(* PLC project SafeLOGIC, BrAutomation SafeDESIGNER  5.24.1.0 *)
(* stored: companyURL http://www.br-automation.com, creationDateTime Tue Nov 25 17:14:16 2025 *)

PROGRAM PARA_INT

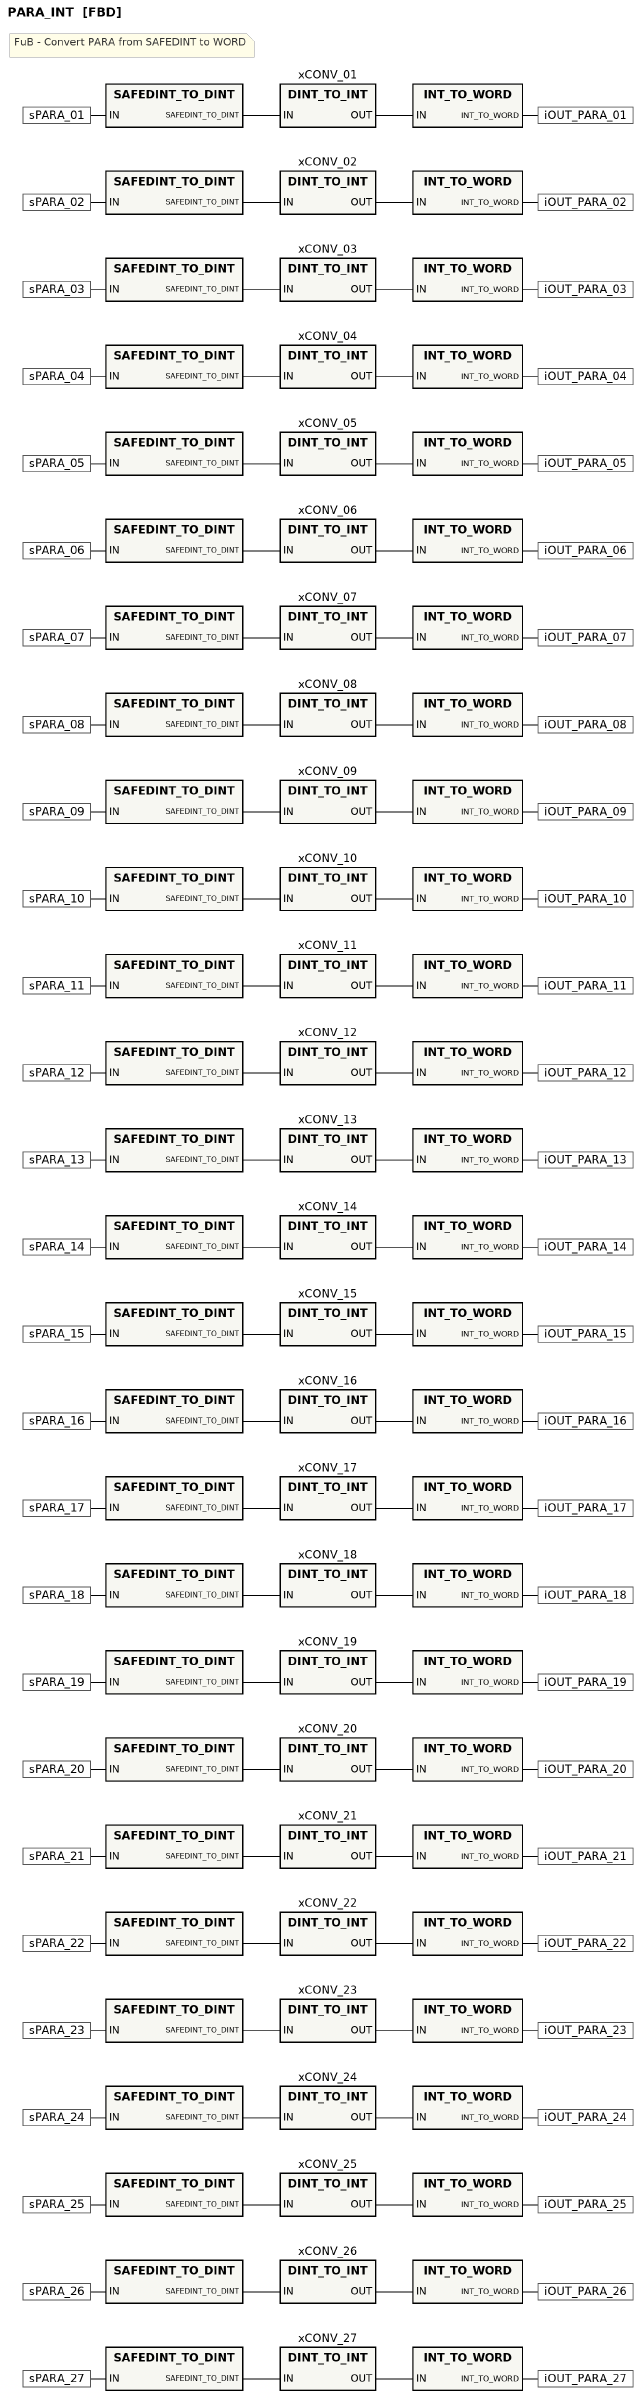
(* FBD diagram, written out as Structured Text *)
(* FuB - Convert PARA from SAFEDINT to WORD *)
xCONV_01(IN := SAFEDINT_TO_DINT(sPARA_01));
iOUT_PARA_01 := INT_TO_WORD(xCONV_01.OUT);
xCONV_02(IN := SAFEDINT_TO_DINT(sPARA_02));
iOUT_PARA_02 := INT_TO_WORD(xCONV_02.OUT);
xCONV_03(IN := SAFEDINT_TO_DINT(sPARA_03));
iOUT_PARA_03 := INT_TO_WORD(xCONV_03.OUT);
xCONV_04(IN := SAFEDINT_TO_DINT(sPARA_04));
iOUT_PARA_04 := INT_TO_WORD(xCONV_04.OUT);
xCONV_05(IN := SAFEDINT_TO_DINT(sPARA_05));
iOUT_PARA_05 := INT_TO_WORD(xCONV_05.OUT);
xCONV_06(IN := SAFEDINT_TO_DINT(sPARA_06));
iOUT_PARA_06 := INT_TO_WORD(xCONV_06.OUT);
xCONV_07(IN := SAFEDINT_TO_DINT(sPARA_07));
iOUT_PARA_07 := INT_TO_WORD(xCONV_07.OUT);
xCONV_08(IN := SAFEDINT_TO_DINT(sPARA_08));
iOUT_PARA_08 := INT_TO_WORD(xCONV_08.OUT);
xCONV_09(IN := SAFEDINT_TO_DINT(sPARA_09));
iOUT_PARA_09 := INT_TO_WORD(xCONV_09.OUT);
xCONV_10(IN := SAFEDINT_TO_DINT(sPARA_10));
iOUT_PARA_10 := INT_TO_WORD(xCONV_10.OUT);
xCONV_11(IN := SAFEDINT_TO_DINT(sPARA_11));
iOUT_PARA_11 := INT_TO_WORD(xCONV_11.OUT);
xCONV_12(IN := SAFEDINT_TO_DINT(sPARA_12));
iOUT_PARA_12 := INT_TO_WORD(xCONV_12.OUT);
xCONV_13(IN := SAFEDINT_TO_DINT(sPARA_13));
iOUT_PARA_13 := INT_TO_WORD(xCONV_13.OUT);
xCONV_14(IN := SAFEDINT_TO_DINT(sPARA_14));
iOUT_PARA_14 := INT_TO_WORD(xCONV_14.OUT);
xCONV_15(IN := SAFEDINT_TO_DINT(sPARA_15));
iOUT_PARA_15 := INT_TO_WORD(xCONV_15.OUT);
xCONV_16(IN := SAFEDINT_TO_DINT(sPARA_16));
iOUT_PARA_16 := INT_TO_WORD(xCONV_16.OUT);
xCONV_17(IN := SAFEDINT_TO_DINT(sPARA_17));
iOUT_PARA_17 := INT_TO_WORD(xCONV_17.OUT);
xCONV_18(IN := SAFEDINT_TO_DINT(sPARA_18));
iOUT_PARA_18 := INT_TO_WORD(xCONV_18.OUT);
xCONV_19(IN := SAFEDINT_TO_DINT(sPARA_19));
iOUT_PARA_19 := INT_TO_WORD(xCONV_19.OUT);
xCONV_20(IN := SAFEDINT_TO_DINT(sPARA_20));
iOUT_PARA_20 := INT_TO_WORD(xCONV_20.OUT);
xCONV_21(IN := SAFEDINT_TO_DINT(sPARA_21));
iOUT_PARA_21 := INT_TO_WORD(xCONV_21.OUT);
xCONV_22(IN := SAFEDINT_TO_DINT(sPARA_22));
iOUT_PARA_22 := INT_TO_WORD(xCONV_22.OUT);
xCONV_23(IN := SAFEDINT_TO_DINT(sPARA_23));
iOUT_PARA_23 := INT_TO_WORD(xCONV_23.OUT);
xCONV_24(IN := SAFEDINT_TO_DINT(sPARA_24));
iOUT_PARA_24 := INT_TO_WORD(xCONV_24.OUT);
xCONV_25(IN := SAFEDINT_TO_DINT(sPARA_25));
iOUT_PARA_25 := INT_TO_WORD(xCONV_25.OUT);
xCONV_26(IN := SAFEDINT_TO_DINT(sPARA_26));
iOUT_PARA_26 := INT_TO_WORD(xCONV_26.OUT);
xCONV_27(IN := SAFEDINT_TO_DINT(sPARA_27));
iOUT_PARA_27 := INT_TO_WORD(xCONV_27.OUT);
END_PROGRAM
